Xinje XCPPro project, PLC1: XC2-42 (software 3.3q)

PROGRAM Ladder

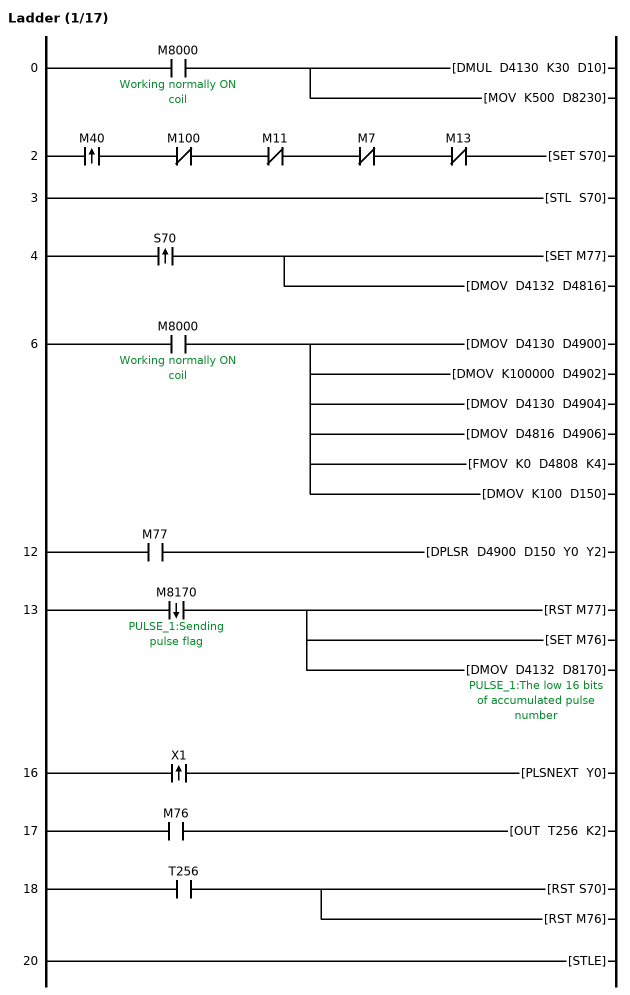
LD     M8000	; Working normally ON coil
DMUL   D4130 K30 D10
MOV    K500 D8230
LDP    M40
ANI    M100
ANI    M11
ANI    M7
ANI    M13
SET    S70
STL    S70
LDP    S70
SET    M77
DMOV   D4132 D4816
LD     M8000	; Working normally ON coil
DMOV   D4130 D4900
DMOV   K100000 D4902
DMOV   D4130 D4904
DMOV   D4816 D4906
FMOV   K0 D4808 K4
DMOV   K100 D150
LD     M77
DPLSR  D4900 D150 Y0 Y2
LDF    M8170	; PULSE_1:Sending pulse flag
RST    M77
SET    M76
DMOV   D4132 D8170	; PULSE_1:The low 16 bits of accumulated pulse number 
LDP    X1
PLSNEXT Y0
LD     M76
OUT    T256 K2
LD     T256
RST    S70
RST    M76
STLE

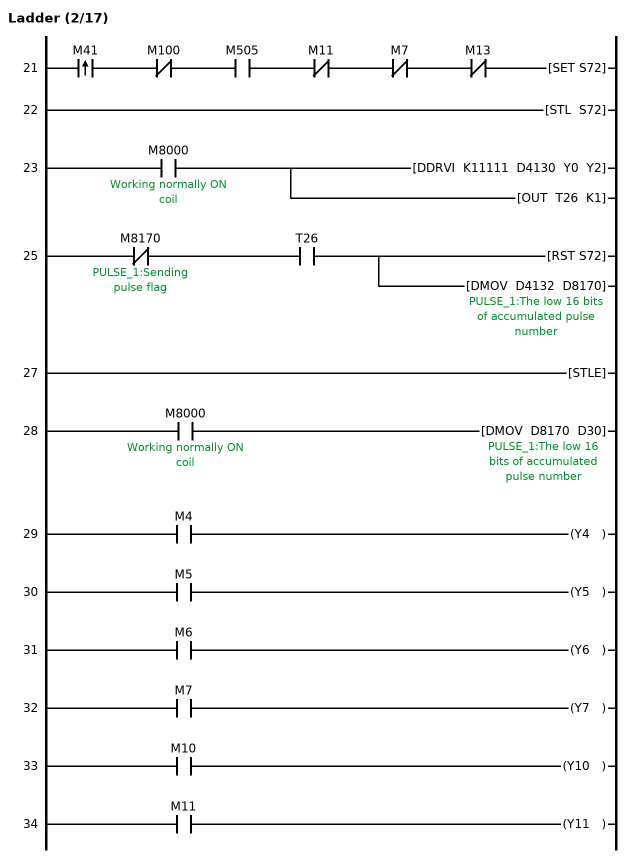
LDP    M41
ANI    M100
AND    M505
ANI    M11
ANI    M7
ANI    M13
SET    S72
STL    S72
LD     M8000	; Working normally ON coil
DDRVI  K11111 D4130 Y0 Y2
OUT    T26 K1
LDI    M8170	; PULSE_1:Sending pulse flag
AND    T26
RST    S72
DMOV   D4132 D8170	; PULSE_1:The low 16 bits of accumulated pulse number 
STLE
LD     M8000	; Working normally ON coil
DMOV   D8170 D30	; PULSE_1:The low 16 bits of accumulated pulse number 
LD     M4
OUT    Y4
LD     M5
OUT    Y5
LD     M6
OUT    Y6
LD     M7
OUT    Y7
LD     M10
OUT    Y10
LD     M11
OUT    Y11

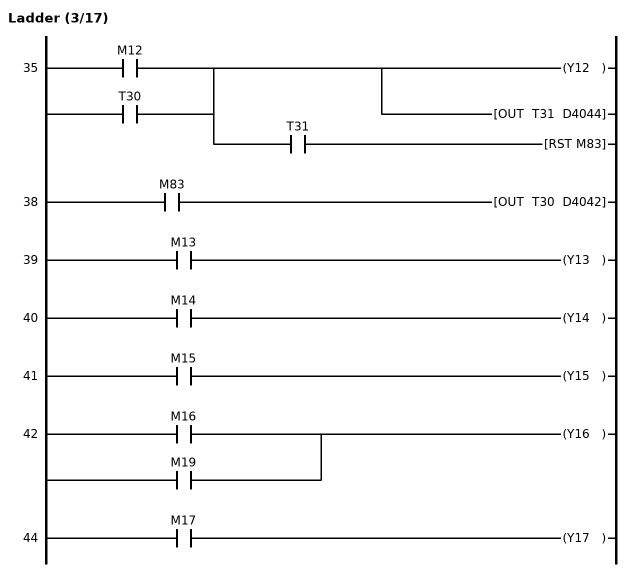
LD     M12
OR     T30
OUT    Y12
OUT    T31 D4044
AND    T31
RST    M83
LD     M83
OUT    T30 D4042
LD     M13
OUT    Y13
LD     M14
OUT    Y14
LD     M15
OUT    Y15
LD     M16
OR     M19
OUT    Y16
LD     M17
OUT    Y17

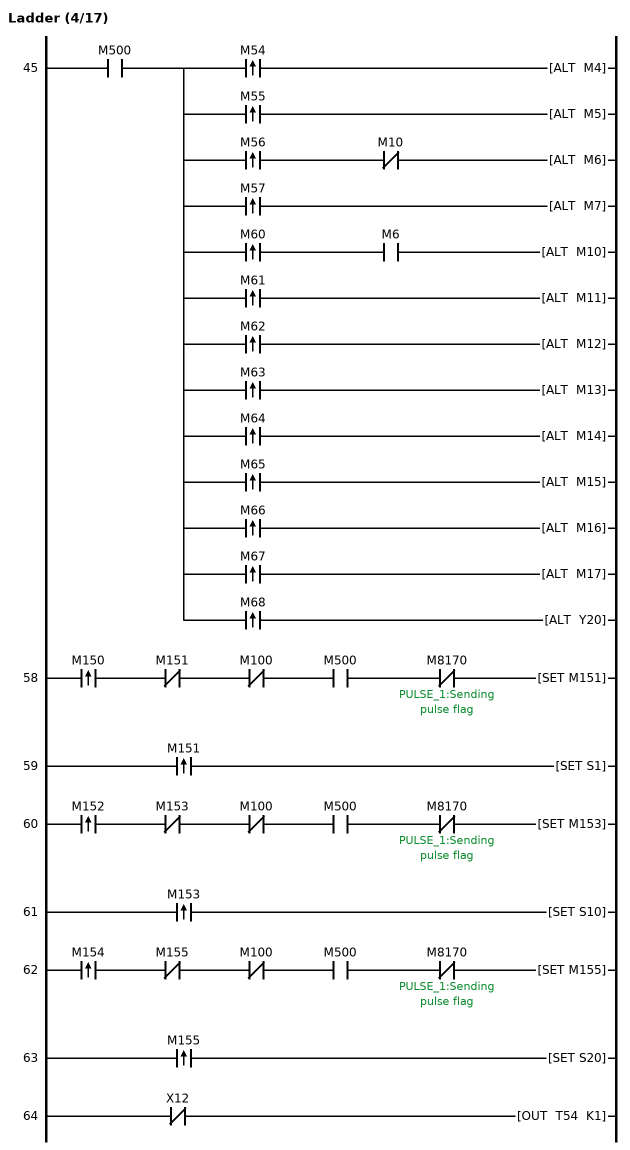
LD     M500
MPS
ANDP   M54
ALT    M4
MRD
ANDP   M55
ALT    M5
MRD
ANDP   M56
ANI    M10
ALT    M6
MRD
ANDP   M57
ALT    M7
MRD
ANDP   M60
AND    M6
ALT    M10
MRD
ANDP   M61
ALT    M11
MRD
ANDP   M62
ALT    M12
MRD
ANDP   M63
ALT    M13
MRD
ANDP   M64
ALT    M14
MRD
ANDP   M65
ALT    M15
MRD
ANDP   M66
ALT    M16
MRD
ANDP   M67
ALT    M17
MPP
ANDP   M68
ALT    Y20
LDP    M150
ANI    M151
ANI    M100
AND    M500
ANI    M8170	; PULSE_1:Sending pulse flag
SET    M151
LDP    M151
SET    S1
LDP    M152
ANI    M153
ANI    M100
AND    M500
ANI    M8170	; PULSE_1:Sending pulse flag
SET    M153
LDP    M153
SET    S10
LDP    M154
ANI    M155
ANI    M100
AND    M500
ANI    M8170	; PULSE_1:Sending pulse flag
SET    M155
LDP    M155
SET    S20
LDI    X12
OUT    T54 K1

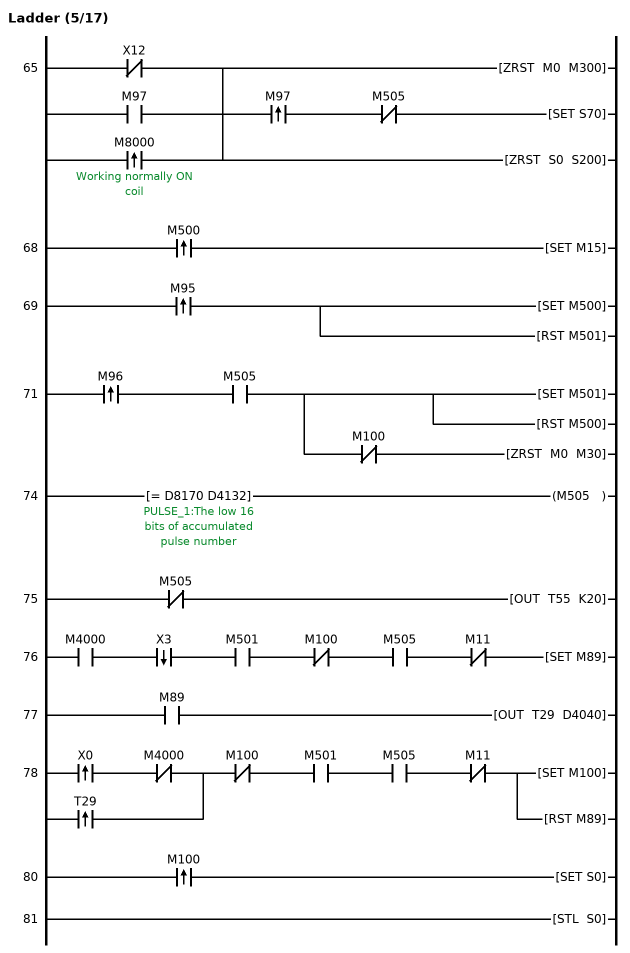
LDI    X12
OR     M97
ORP    M8000	; Working normally ON coil
ZRST   M0 M300
MPS
ANDP   M97
ANI    M505
SET    S70
MPP
ZRST   S0 S200
LDP    M500
SET    M15
LDP    M95
SET    M500
RST    M501
LDP    M96
AND    M505
SET    M501
RST    M500
ANI    M100
ZRST   M0 M30
LD=    D8170 D4132	; PULSE_1:The low 16 bits of accumulated pulse number 
OUT    M505
LDI    M505
OUT    T55 K20
LD     M4000
ANDF   X3
AND    M501
ANI    M100
AND    M505
ANI    M11
SET    M89
LD     M89
OUT    T29 D4040
LDP    X0
ANI    M4000
ORP    T29
ANI    M100
AND    M501
AND    M505
ANI    M11
SET    M100
RST    M89
LDP    M100
SET    S0
STL    S0

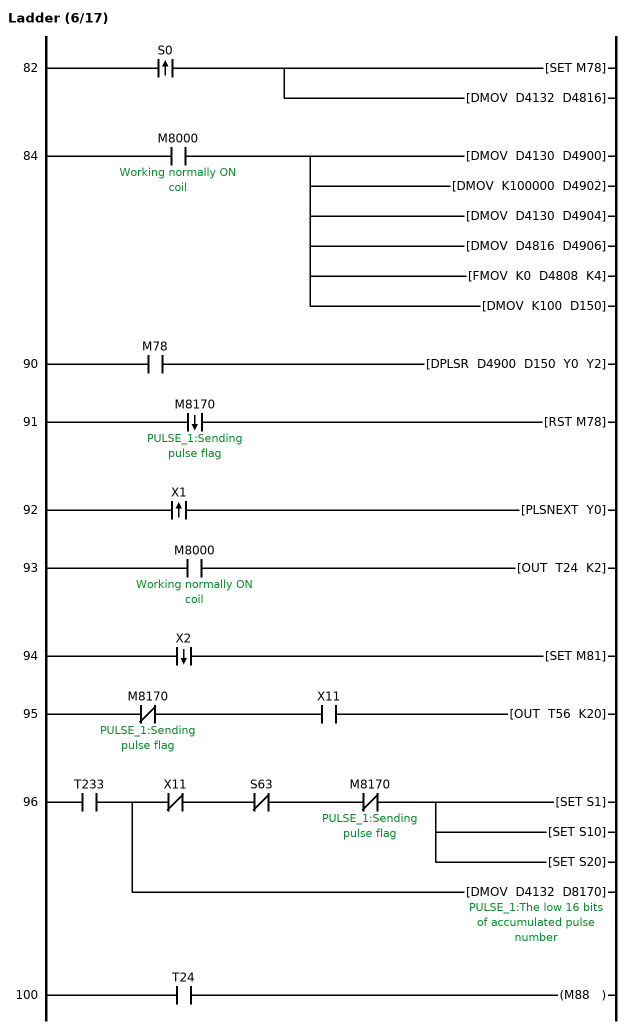
LDP    S0
SET    M78
DMOV   D4132 D4816
LD     M8000	; Working normally ON coil
DMOV   D4130 D4900
DMOV   K100000 D4902
DMOV   D4130 D4904
DMOV   D4816 D4906
FMOV   K0 D4808 K4
DMOV   K100 D150
LD     M78
DPLSR  D4900 D150 Y0 Y2
LDF    M8170	; PULSE_1:Sending pulse flag
RST    M78
LDP    X1
PLSNEXT Y0
LD     M8000	; Working normally ON coil
OUT    T24 K2
LDF    X2
SET    M81
LDI    M8170	; PULSE_1:Sending pulse flag
AND    X11
OUT    T56 K20
LD     T233
MPS
ANI    X11
ANI    S63
ANI    M8170	; PULSE_1:Sending pulse flag
SET    S1
SET    S10
SET    S20
MPP
DMOV   D4132 D8170	; PULSE_1:The low 16 bits of accumulated pulse number 
LD     T24
OUT    M88

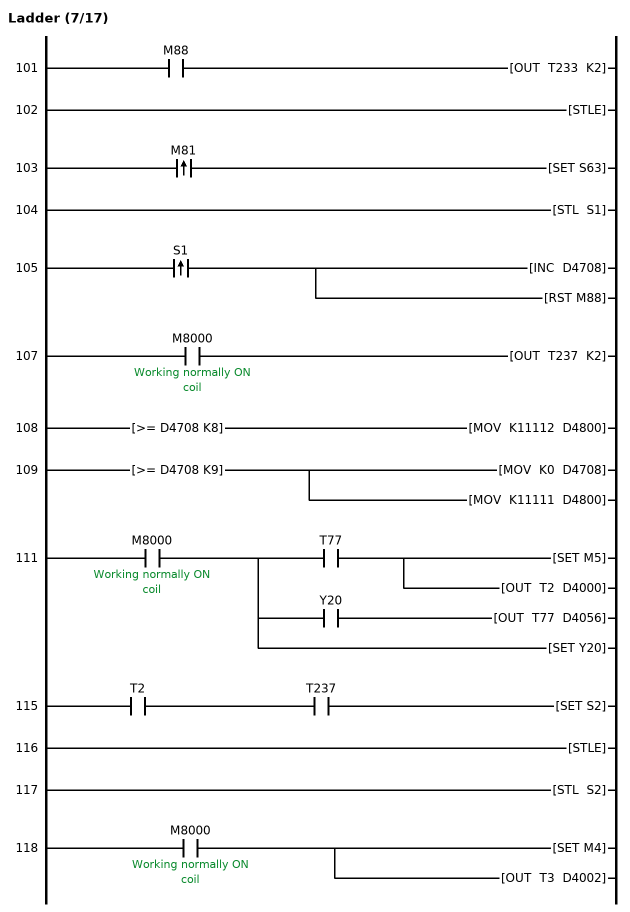
LD     M88
OUT    T233 K2
STLE
LDP    M81
SET    S63
STL    S1
LDP    S1
INC    D4708
RST    M88
LD     M8000	; Working normally ON coil
OUT    T237 K2
LD>=   D4708 K8
MOV    K11112 D4800
LD>=   D4708 K9
MOV    K0 D4708
MOV    K11111 D4800
LD     M8000	; Working normally ON coil
MPS
AND    T77
SET    M5
OUT    T2 D4000
MRD
AND    Y20
OUT    T77 D4056
MPP
SET    Y20
LD     T2
AND    T237
SET    S2
STLE
STL    S2
LD     M8000	; Working normally ON coil
SET    M4
OUT    T3 D4002

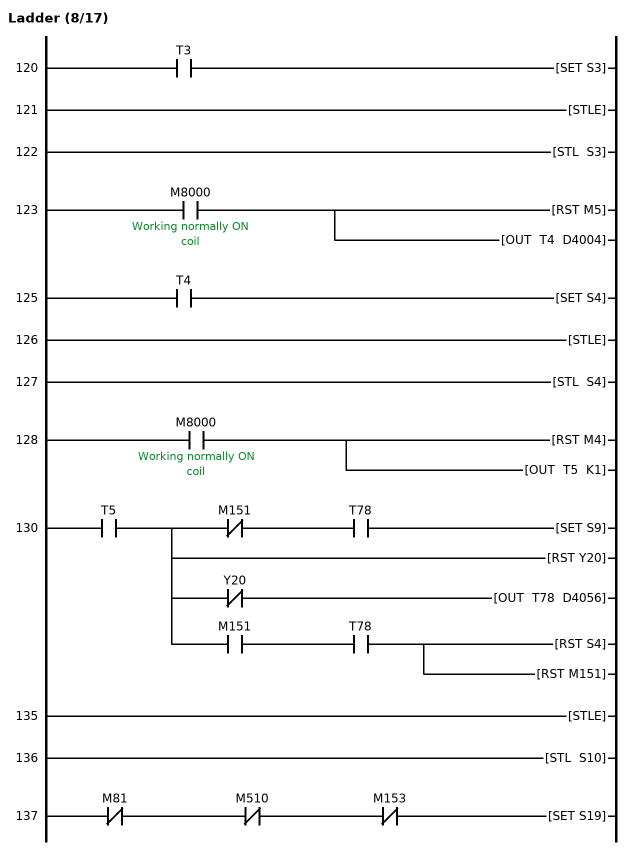
LD     T3
SET    S3
STLE
STL    S3
LD     M8000	; Working normally ON coil
RST    M5
OUT    T4 D4004
LD     T4
SET    S4
STLE
STL    S4
LD     M8000	; Working normally ON coil
RST    M4
OUT    T5 K1
LD     T5
MPS
ANI    M151
AND    T78
SET    S9
MRD
RST    Y20
ANI    Y20
OUT    T78 D4056
MPP
AND    M151
AND    T78
RST    S4
RST    M151
STLE
STL    S10
LDI    M81
ANI    M510
ANI    M153
SET    S19

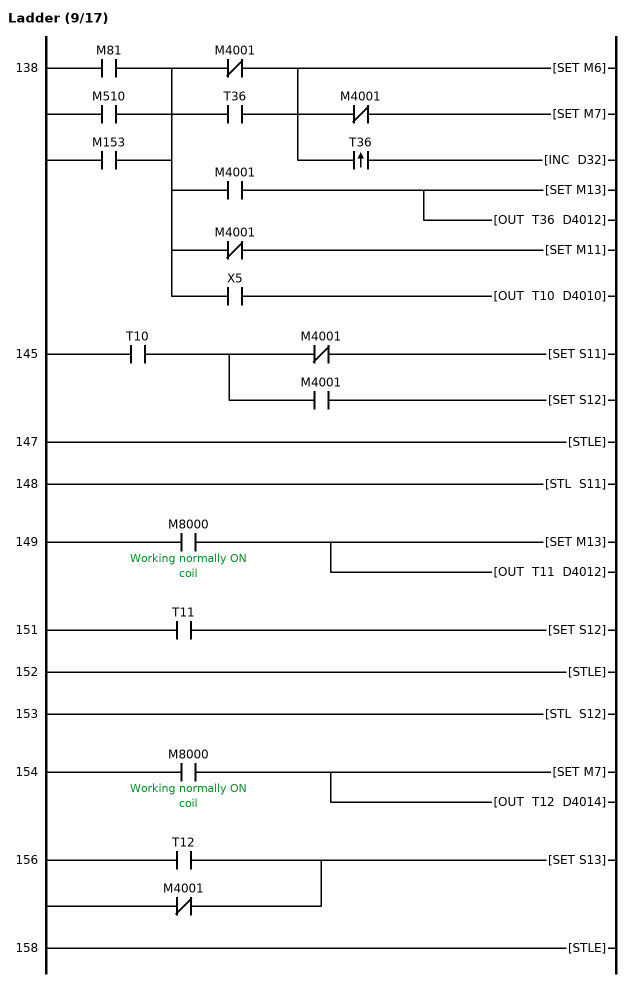
LD     M81
OR     M510
OR     M153
MPS
LDI    M4001
OR     T36
ANB
SET    M6
MPS
ANI    M4001
SET    M7
MPP
ANDP   T36
INC    D32
MRD
AND    M4001
SET    M13
OUT    T36 D4012
MRD
ANI    M4001
SET    M11
MPP
AND    X5
OUT    T10 D4010
LD     T10
MPS
ANI    M4001
SET    S11
MPP
AND    M4001
SET    S12
STLE
STL    S11
LD     M8000	; Working normally ON coil
SET    M13
OUT    T11 D4012
LD     T11
SET    S12
STLE
STL    S12
LD     M8000	; Working normally ON coil
SET    M7
OUT    T12 D4014
LD     T12
ORI    M4001
SET    S13
STLE

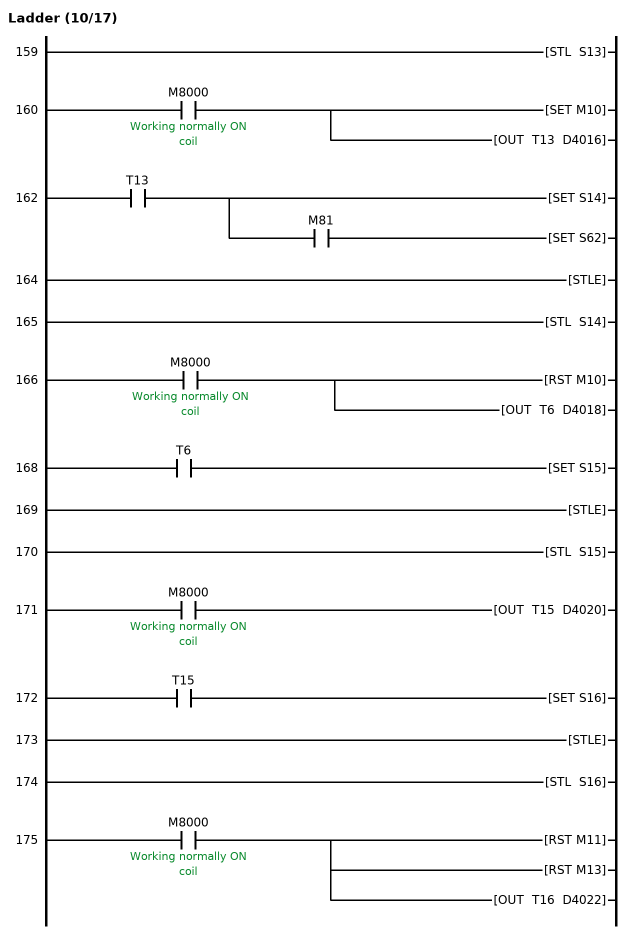
STL    S13
LD     M8000	; Working normally ON coil
SET    M10
OUT    T13 D4016
LD     T13
SET    S14
AND    M81
SET    S62
STLE
STL    S14
LD     M8000	; Working normally ON coil
RST    M10
OUT    T6 D4018
LD     T6
SET    S15
STLE
STL    S15
LD     M8000	; Working normally ON coil
OUT    T15 D4020
LD     T15
SET    S16
STLE
STL    S16
LD     M8000	; Working normally ON coil
RST    M11
RST    M13
OUT    T16 D4022

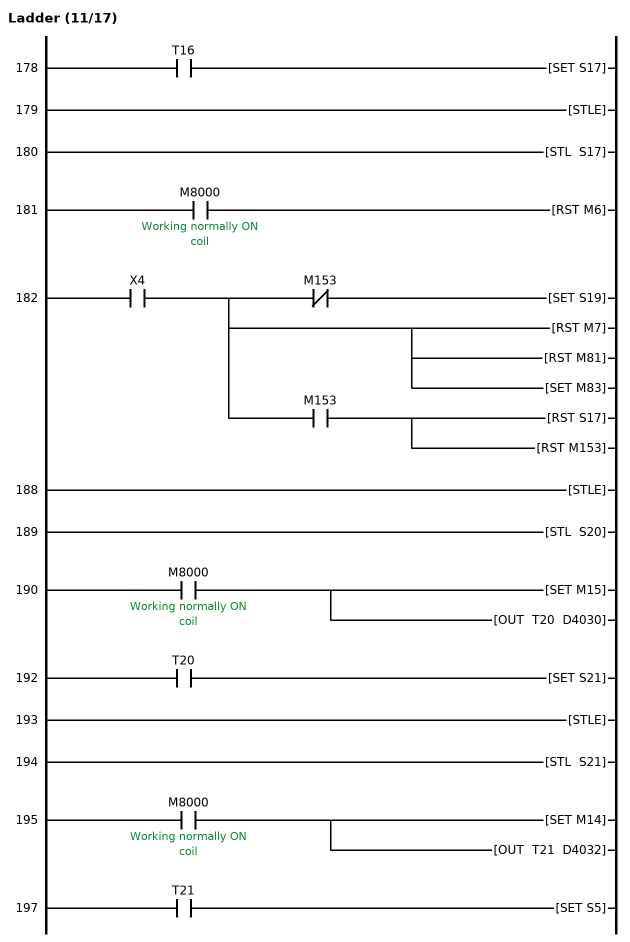
LD     T16
SET    S17
STLE
STL    S17
LD     M8000	; Working normally ON coil
RST    M6
LD     X4
MPS
ANI    M153
SET    S19
MPP
RST    M7
RST    M81
SET    M83
AND    M153
RST    S17
RST    M153
STLE
STL    S20
LD     M8000	; Working normally ON coil
SET    M15
OUT    T20 D4030
LD     T20
SET    S21
STLE
STL    S21
LD     M8000	; Working normally ON coil
SET    M14
OUT    T21 D4032
LD     T21
SET    S5

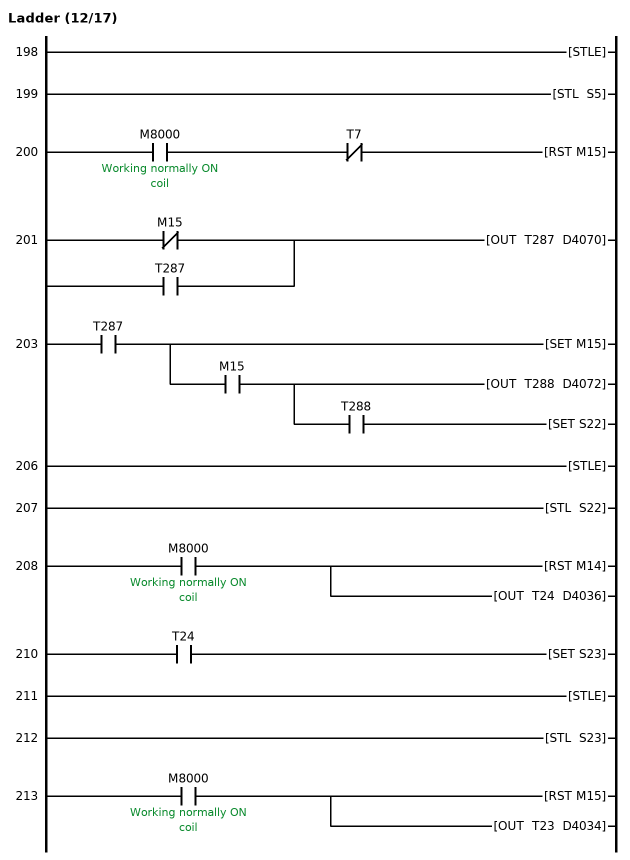
STLE
STL    S5
LD     M8000	; Working normally ON coil
ANI    T7
RST    M15
LDI    M15
OR     T287
OUT    T287 D4070
LD     T287
SET    M15
AND    M15
OUT    T288 D4072
AND    T288
SET    S22
STLE
STL    S22
LD     M8000	; Working normally ON coil
RST    M14
OUT    T24 D4036
LD     T24
SET    S23
STLE
STL    S23
LD     M8000	; Working normally ON coil
RST    M15
OUT    T23 D4034

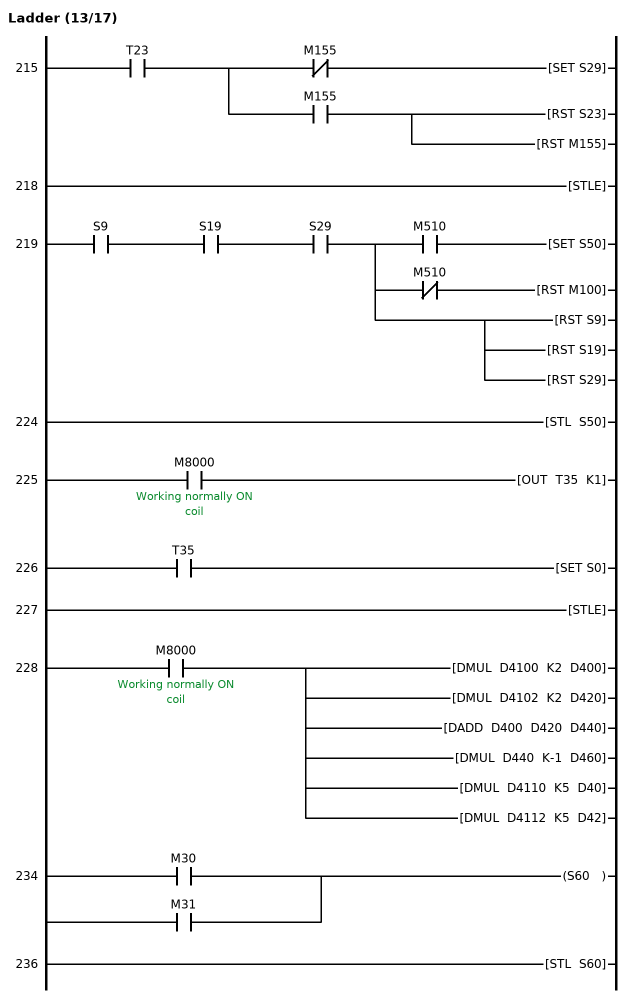
LD     T23
MPS
ANI    M155
SET    S29
MPP
AND    M155
RST    S23
RST    M155
STLE
LD     S9
AND    S19
AND    S29
MPS
AND    M510
SET    S50
MRD
ANI    M510
RST    M100
MPP
RST    S9
RST    S19
RST    S29
STL    S50
LD     M8000	; Working normally ON coil
OUT    T35 K1
LD     T35
SET    S0
STLE
LD     M8000	; Working normally ON coil
DMUL   D4100 K2 D400
DMUL   D4102 K2 D420
DADD   D400 D420 D440
DMUL   D440 K-1 D460
DMUL   D4110 K5 D40
DMUL   D4112 K5 D42
LD     M30
OR     M31
OUT    S60
STL    S60

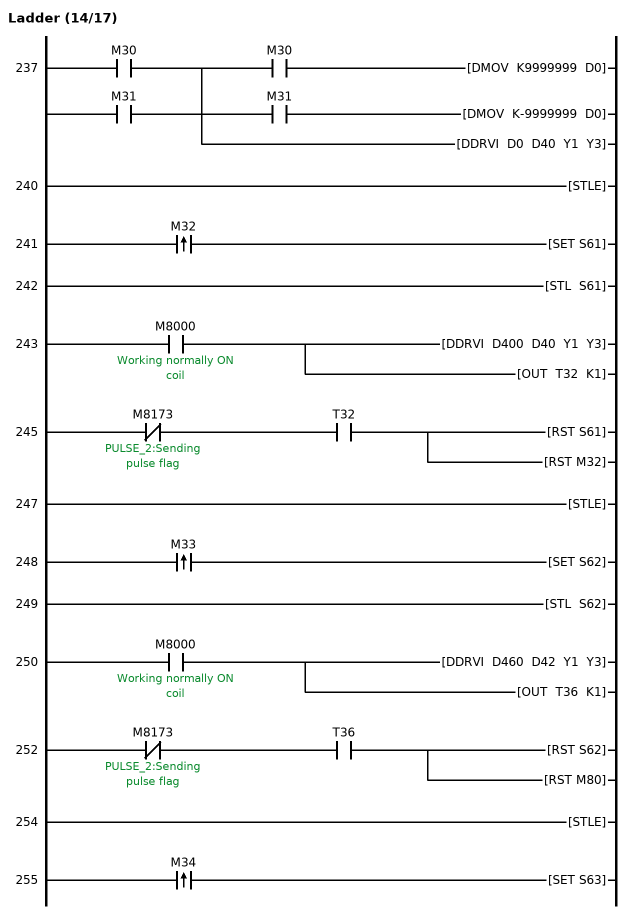
LD     M30
OR     M31
MPS
AND    M30
DMOV   K9999999 D0
MRD
AND    M31
DMOV   K-9999999 D0
MPP
DDRVI  D0 D40 Y1 Y3
STLE
LDP    M32
SET    S61
STL    S61
LD     M8000	; Working normally ON coil
DDRVI  D400 D40 Y1 Y3
OUT    T32 K1
LDI    M8173	; PULSE_2:Sending pulse flag
AND    T32
RST    S61
RST    M32
STLE
LDP    M33
SET    S62
STL    S62
LD     M8000	; Working normally ON coil
DDRVI  D460 D42 Y1 Y3
OUT    T36 K1
LDI    M8173	; PULSE_2:Sending pulse flag
AND    T36
RST    S62
RST    M80
STLE
LDP    M34
SET    S63

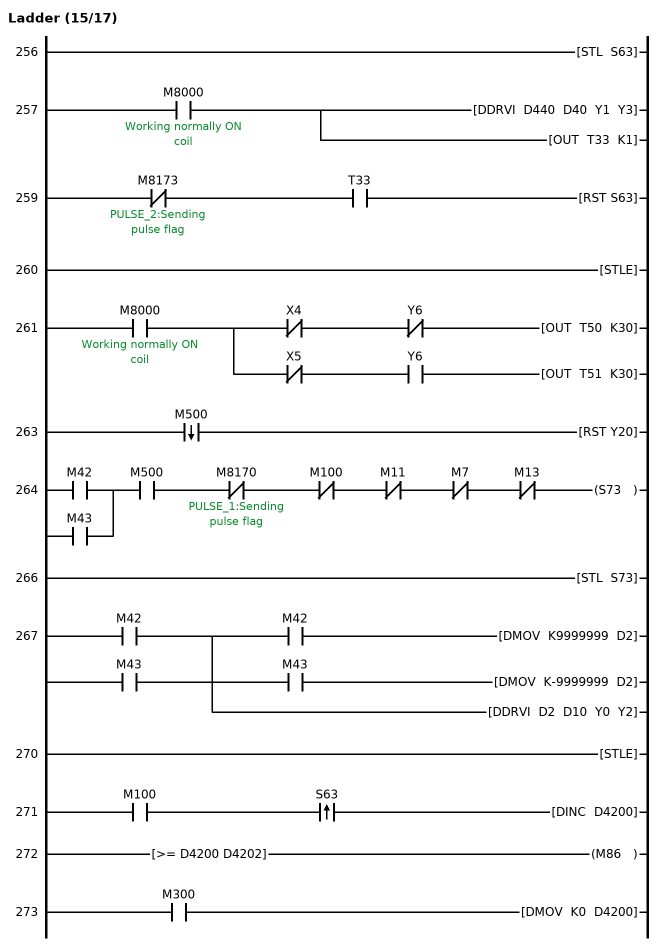
STL    S63
LD     M8000	; Working normally ON coil
DDRVI  D440 D40 Y1 Y3
OUT    T33 K1
LDI    M8173	; PULSE_2:Sending pulse flag
AND    T33
RST    S63
STLE
LD     M8000	; Working normally ON coil
MPS
ANI    X4
ANI    Y6
OUT    T50 K30
MPP
ANI    X5
AND    Y6
OUT    T51 K30
LDF    M500
RST    Y20
LD     M42
OR     M43
AND    M500
ANI    M8170	; PULSE_1:Sending pulse flag
ANI    M100
ANI    M11
ANI    M7
ANI    M13
OUT    S73
STL    S73
LD     M42
OR     M43
MPS
AND    M42
DMOV   K9999999 D2
MRD
AND    M43
DMOV   K-9999999 D2
MPP
DDRVI  D2 D10 Y0 Y2
STLE
LD     M100
ANDP   S63
DINC   D4200
LD>=   D4200 D4202
OUT    M86
LD     M300
DMOV   K0 D4200

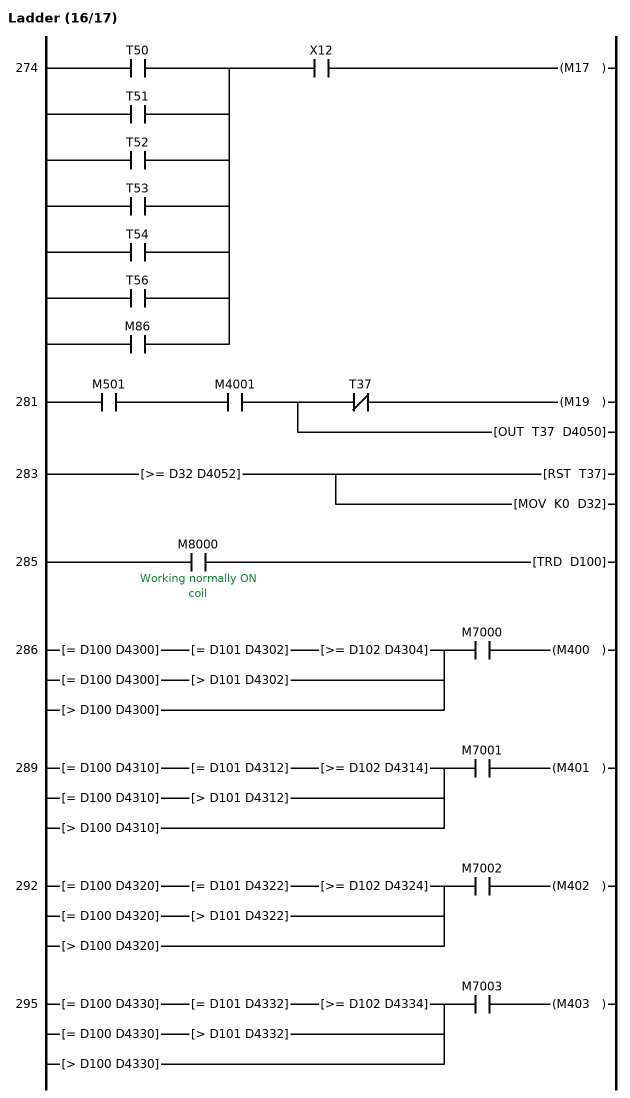
LD     T50
OR     T51
OR     T52
OR     T53
OR     T54
OR     T56
OR     M86
AND    X12
OUT    M17
LD     M501
AND    M4001
MPS
ANI    T37
OUT    M19
MPP
OUT    T37 D4050
LD>=   D32 D4052
RST    T37
MOV    K0 D32
LD     M8000	; Working normally ON coil
TRD    D100
LD=    D100 D4300
AND=   D101 D4302
AND>=  D102 D4304
LD=    D100 D4300
AND>   D101 D4302
ORB
OR>    D100 D4300
AND    M7000
OUT    M400
LD=    D100 D4310
AND=   D101 D4312
AND>=  D102 D4314
LD=    D100 D4310
AND>   D101 D4312
ORB
OR>    D100 D4310
AND    M7001
OUT    M401
LD=    D100 D4320
AND=   D101 D4322
AND>=  D102 D4324
LD=    D100 D4320
AND>   D101 D4322
ORB
OR>    D100 D4320
AND    M7002
OUT    M402
LD=    D100 D4330
AND=   D101 D4332
AND>=  D102 D4334
LD=    D100 D4330
AND>   D101 D4332
ORB
OR>    D100 D4330
AND    M7003
OUT    M403

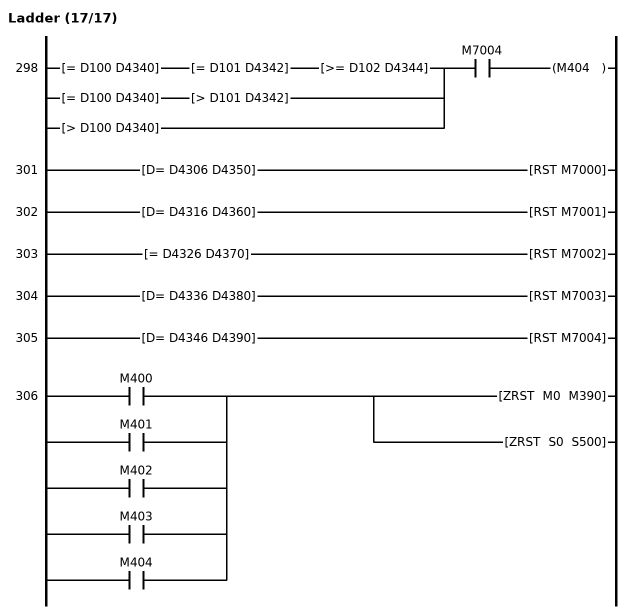
LD=    D100 D4340
AND=   D101 D4342
AND>=  D102 D4344
LD=    D100 D4340
AND>   D101 D4342
ORB
OR>    D100 D4340
AND    M7004
OUT    M404
DLD=   D4306 D4350
RST    M7000
DLD=   D4316 D4360
RST    M7001
LD=    D4326 D4370
RST    M7002
DLD=   D4336 D4380
RST    M7003
DLD=   D4346 D4390
RST    M7004
LD     M400
OR     M401
OR     M402
OR     M403
OR     M404
ZRST   M0 M390
ZRST   S0 S500